% RSLogix 500 project myPlc.RSS, saved by version 8.40.00.08 %
PROJECT "MYPLC"    % processor: Bul.1763 MicroLogix 1100 Series A %

PROGRAM FILES
  LAD 2   7 rungs

DATA FILES
  O0 OUTPUT  4 elements
  I1 INPUT  6 elements
  S2 STATUS  66 elements
  B3 BINARY  1 elements
  T4 TIMER  1 elements
  C5 COUNTER  1 elements
  R6 CONTROL  1 elements
  N7 INTEGER  1 elements
  F8 FLOAT  1 elements

LADDER 2
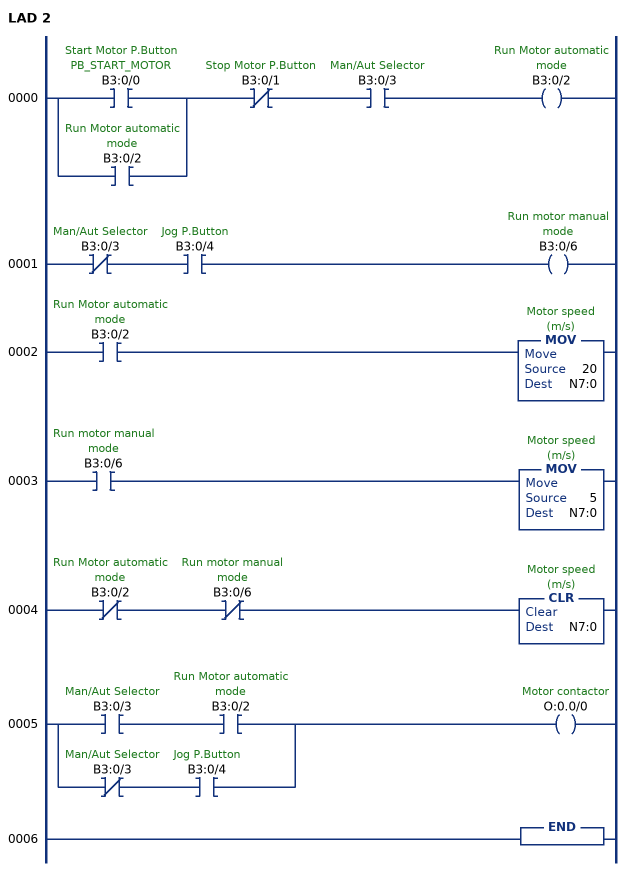
% Rung: 0 %
SOR BST XIC B3:0/0 NXB XIC B3:0/2 BND XIO B3:0/1 XIC B3:0/3 OTE B3:0/2 EOR
%   B3:0/0  PB_START_MOTOR  "Start Motor P.Button" %
%   B3:0/2  "Run Motor automatic mode" %
%   B3:0/1  "Stop Motor P.Button" %
%   B3:0/3  "Man/Aut Selector" %
% Rung: 1 %
SOR XIO B3:0/3 XIC B3:0/4 OTE B3:0/6 EOR
%   B3:0/3  "Man/Aut Selector" %
%   B3:0/4  "Jog P.Button" %
%   B3:0/6  "Run motor manual mode" %
% Rung: 2 %
SOR XIC B3:0/2 MOV 20 N7:0 EOR
%   B3:0/2  "Run Motor automatic mode" %
%   N7:0  "Motor speed (m/s)" %
% Rung: 3 %
SOR XIC B3:0/6 MOV 5 N7:0 EOR
%   B3:0/6  "Run motor manual mode" %
%   N7:0  "Motor speed (m/s)" %
% Rung: 4 %
SOR XIO B3:0/2 XIO B3:0/6 CLR N7:0 EOR
%   B3:0/2  "Run Motor automatic mode" %
%   B3:0/6  "Run motor manual mode" %
%   N7:0  "Motor speed (m/s)" %
% Rung: 5 %
SOR BST XIC B3:0/3 XIC B3:0/2 NXB XIO B3:0/3 XIC B3:0/4 BND OTE O:0.0/0 EOR
%   B3:0/3  "Man/Aut Selector" %
%   B3:0/2  "Run Motor automatic mode" %
%   B3:0/4  "Jog P.Button" %
%   O:0.0/0  "Motor contactor" %
% Rung: 6 %
SOR END EOR

OTHER DOCUMENTED ADDRESSES
  B3:0/5  "Jog Motor"
